TYPE ST_Auto_UpperFeedInConveyor :
STRUCT
	Command		: ST_Auto_UpperFeedInConveyorCommand;
	Status		: ST_Auto_UpperFeedInConveyorStatus;	
	Info		: ST_Auto_UpperFeedInConveyorInfo;
	FeedBack    : ST_Auto_UpperFeedInConveyorFeedback;	
	
END_STRUCT
END_TYPE

(* stored: Version 1.1.0.1, ProductVersion 3.1.4024.13
   DUT ST_Auto_UpperFeedInConveyor: Id {f7a64b28-0d6b-4704-860e-e477f3bc1ee5} *)
